FUNCTION F_LogA5 
VAR_INPUT
	eLogLevel		: E_LogLevel;
	sMessage		: T_MaxString;
	aArg1			: ANY;
	aArg2			: ANY;
	aArg3			: ANY;
	aArg4			: ANY;
	aArg5			: ANY;
END_VAR

F_LogLA5(eLogLevel, Const.sGlobalLogger, sMessage, aArg1, aArg2, aArg3, aArg4, aArg5);

END_FUNCTION

(* stored: Version 1.1.0.1, ProductVersion 3.1.4024.0
   POU F_LogA5: Id {85bfdb20-ca04-4e2e-8d69-7de901c475f4}, SpecialFunc None *)
